//==================================================================================================
//							Beckhoff Automation Poland
//									12.04.2018
//	Blok funkcyjny kontroli luzownika w silniku podpietym do AX8000. Przewaga ForceLock
//	Dzialania na obiekcie: 3000:07 Motor brake force
//	Index:			AxisMainSlot: 16#3000 (Ch A)/ 16#3400 (Ch B)
//	Subindex:		16#07
//	Datatype:		ENUM (INT16)
//	Enum Value:		0 (0x00): 	Release_force
//					1 (0x01): 	Force_lock
//					2 (0x02): 	Force_unlock
//
//  v1.0	|| TC v 3.1.4022.16		|| - pierwsza wersja
//==================================================================================================
FUNCTION_BLOCK FB_HoldingBrakeCtrlAX8000_1
VAR_INPUT
	bForceLock 						: BOOL;								// 
	bForceUnlock					: BOOL;								// 
	stDriveRef						: ST_DriveRef;
END_VAR
VAR_OUTPUT
	bBusy							: BOOL;
	bError							: BOOL; 							// General error: parameter or CoE read.
																		// If bError = TRUE and bInitialized = FALSE - error during read motor data.
																		// If bError = TRUE and bInitialized = TRUE and (iAdsErrId <> 0 or iCANopenErrId <> 0) then I2T read error
																		// If bError = TRUE and bInitialized = TRUE and iAdsErrId = 0 and iCANopenErrId = 0 then parameter error: rTorqueLimit outside permitted range rTorqueLimitLow..rTorqueLimitHigh or Empty stDriveRef
	iAdsErrId						: UINT;								// Forwarded output FB_CoERead_ByDriveRef
	iCANopenErrId					: UINT;								// Forwarded output FB_CoERead_ByDriveRef
END_VAR
VAR
	bExecute						: BOOL;
	iMotorBrakeForce				: INT;								// 0 - Release_force, 1 - Force_lock, 2 - Force_unlock
	rtForceLock						: R_TRIG;
	rtForceUnlock					: R_TRIG;
	ftForceLock						: F_TRIG;
	ftForceUnlock					: F_TRIG;
	fbForceLockUnlock				: FB_CoEWrite_ByDriveRef;
END_VAR

{region "Call triggers"}
//======================= Call triggers =========================
rtForceLock(CLK:= bForceLock);
ftForceLock(CLK:= bForceLock);
rtForceUnlock(CLK:= bForceUnlock);
ftForceUnlock(CLK:= bForceUnlock);
bExecute								:= rtForceLock.Q OR ftForceLock.Q OR rtForceUnlock.Q OR ftForceUnlock.Q;
//===============================================================
{endregion}
{region "Main code"}
//========================= Main code ===========================
IF bExecute THEN
	iMotorBrakeForce 						:= 0;										// Clear value
	iMotorBrakeForce.1 						:= bForceUnlock;							// Set force unlock bit
	iMotorBrakeForce 						:= SEL(bForceLock, iMotorBrakeForce, 1);	// Set force lock bit, it has higher priority than unlock
END_IF

fbForceLockUnlock(	stDriveRef				:= stDriveRef, 
					nIndex					:= 16#3000 + (stDriveRef.nDriveNo * 16#400), 
					nSubIndex				:= 16#07, 
					pSrcBuf					:= ADR(iMotorBrakeForce), 
					cbBufLen				:= SIZEOF(iMotorBrakeForce), 
					bExecute				:= bExecute,
					bBusy					=> bBusy, 
					bError					=> bError, 
					iAdsErrId				=> iAdsErrId, 
					iCANopenErrId			=> iCANopenErrId);
//===============================================================
{endregion}

END_FUNCTION_BLOCK

(* stored: Version 1.2.0.0, ProductVersion 3.1.4026.13, FileIdentifier 870f01acbae856811fd15ce5150ea9764ca3b016, FileSignature 0f739d15884e1e887f19e32a62a01f3135159cc530433a2fffd774076629df56ba54b4fffe4b2eeb681bbc92b509631db3ef242d38fc132a30201ddd5cae816b7dcf14e1ab4421f9aa3c645590827134f6b5066a0f2722663eb3d8fdd4aee54d09a1b4f0f1649ee74bebd92e745aeccd04213b6321e14628b2989db022dfe7c58120ffef5f29c70dbf691768dbd51a7b73d7c68b7254e06807a7d74beb93484927c5f0329cb8413c73b81b72485df25b487aede2315166d209001478e9b1bbf37ed8696b267cfba6d5e8966a509c8d07f08262bcee1395480a89215644bbb4a607ec0abd63dcdefebfb1932c5c21c81f6aa57befe52329c6bb0e642aadc77c42
   POU FB_HoldingBrakeCtrlAX8000_1: Id {9552c8d8-3f9e-48b3-a8ab-bbc016235e03}, SpecialFunc None *)
